FUNCTION_BLOCK EcMasterGetAbnortalStateChange IMPLEMENTS IEcTask
VAR_INPUT
END_VAR
VAR_OUTPUT
END_VAR
VAR
	iState : INT;
	masterAbnormalStateChanges : Tc2_EtherCAT.FB_EcGetAllSlaveAbnormalStateChanges;
	_abnormalStates : ARRAY[0..Tc2_EtherCAT.EC_MAX_SLAVES] OF UDINT;
	_execute: BOOL;
	_done: BOOL;
	_busy: BOOL;
	_error: BOOL;
	_netId: AMSNETID;
END_VAR

CASE iState OF
	0:
		IF _execute THEN
			_done := FALSE;
			_busy := TRUE;
			_error := FALSE;
			masterAbnormalStateChanges.bExecute := TRUE;
			IF masterAbnormalStateChanges.bBusy THEN
				iState := 10;
				_execute := false;
			END_IF
		END_IF
	10:
		IF NOT masterAbnormalStateChanges.bBusy THEN
			IF NOT masterAbnormalStateChanges.bError THEN
				_done := TRUE;
			ELSE
				_error := TRUE;
			END_IF
			_busy := FALSE;
			masterAbnormalStateChanges.bExecute := FALSE;
			iState := 0;
		END_IF
END_CASE

masterAbnormalStateChanges(sNetId := Tc2_System.F_CreateAmsNetId(nIds := NetId),
							pAddrBuf := ADR(_abnormalStates),
							cbBufLen := SIZEOF(_abnormalStates));

PROPERTY AbnormalStateChanges : reference to array[0..EC_MAX_Slaves] of udint
GET
AbnormalStateChanges REF= _abnormalStates;
END_GET
END_PROPERTY

{warning 'add method implementation '}
METHOD Abort : BOOL
masterAbnormalStateChanges.bExecute := FALSE;
_busy := FALSE;
_execute := FALSE;
Abort := TRUE;
iState := 0;
END_METHOD

{warning 'add property implementation'}
PROPERTY Busy : BOOL
GET
Busy := _busy;
END_GET
END_PROPERTY

{warning 'add property implementation'}
PROPERTY Done : BOOL
GET
Done := _done;
END_GET
END_PROPERTY

{warning 'add property implementation'}
PROPERTY Error : BOOL
GET
Error := _error;
END_GET
END_PROPERTY

{warning 'add method implementation '}
METHOD Execute : BOOL
IF NOT masterAbnormalStateChanges.bBusy THEN
	Execute := _execute := true;
END_IF
END_METHOD

{warning 'add property implementation'}
PROPERTY NetID : amsnetid
GET
NetID := _netId;
END_GET
SET
_netId := NetID;
END_SET
END_PROPERTY

END_FUNCTION_BLOCK

(* stored: Version 1.1.0.1, ProductVersion 3.1.4024.11
   POU EcMasterGetAbnortalStateChange: Id {916ca048-2a5d-4fdb-b2cb-ddd18890c471}, SpecialFunc None
   Property AbnormalStateChanges: Id {47a02964-f488-4b9c-809a-d7ee720640e6}
   Get Get: Id {014b0af4-0de3-4019-9f68-81183b1f6216}
   Method Abort: Id {1f265fd5-2b4f-4969-96fd-1a379195b145}
   Property Busy: Id {e8d03f9f-63f3-428a-8de6-e9e691304f77}
   Get Get: Id {564ae041-99a6-46e5-ae6c-5eb1730e0a8f}
   Property Done: Id {23568b10-02d3-4e4f-84a4-ef7d3bbb49a4}
   Get Get: Id {aa3eec7b-376c-4c4e-b565-461d43b331d2}
   Property Error: Id {b1c9d995-aca8-469c-96dd-255610ef94f0}
   Get Get: Id {76f43c01-ba0b-4500-95ec-2257af077f54}
   Method Execute: Id {43b79ca5-25c4-4be4-aab3-772100dcd003}
   Property NetID: Id {875224f8-a4d2-433a-a701-440c539aef98}
   Get Get: Id {96282c8d-4aaa-4d0a-b3e2-1f8590fdbc0b}
   Set Set: Id {7411c9b2-9fdb-4474-9c62-eba9418dcc1d} *)
